TYPE ST_IoT_Device_General :
STRUCT

	sDeviceName					: STRING;	
	sDeviceIcon					: STRING;
	sMainTopic					: STRING;
	
END_STRUCT
END_TYPE

(* stored: Version 1.1.0.1, ProductVersion 3.1.4024.12
   DUT ST_IoT_Device_General: Id {efd5a8b1-fa6e-4081-a6a7-ba4a2a80bbec} *)
